(* IEC 61131-3 sources: repolevel_ST_code_completion/output/0127完整版本_带planner/repoeval_Command1/readful_result_no_provide, 10 files *)

(* ---- FB_AirConditioning.st ---- *)
FUNCTION_BLOCK PUBLIC FB_AirConditioning
VAR_OUTPUT
bActive			: BOOL;
lrTemperature	: LREAL;
END_VAR
VAR
lrDefaultTemperature : LREAL := LREAL#0.0; // Explicitly typed initialization
lrCalculatedTemperature : LREAL;
END_VAR

IF bActive THEN
// Calculate the current environment temperature based on control logic
lrCalculatedTemperature := 23.5; // Example fixed value, as logic isn't provided
lrTemperature := lrCalculatedTemperature;
ELSE
// Set temperature to default value when inactive
lrTemperature := lrDefaultTemperature;
END_IF

END_FUNCTION_BLOCK

(* ---- FB_Lamp.st ---- *)
FUNCTION_BLOCK PUBLIC FB_Lamp
VAR_OUTPUT
  byLevel			: BYTE;
END_VAR
VAR
  byNewLevel		: BYTE;
END_VAR

IF byNewLevel > 255 THEN
  byLevel := 255;
ELSE
  byLevel := byNewLevel;
END_IF;
END_FUNCTION_BLOCK

(* ---- FB_Socket.st ---- *)
FUNCTION_BLOCK FB_Socket
VAR_OUTPUT
bActive		: BOOL;
END_VAR
VAR
bInitialized : BOOL := FALSE;
bConnected   : BOOL := FALSE;
END_VAR

IF NOT bInitialized THEN
(* Initialize the socket *)
bInitialized := TRUE;
(* bConnected remains as FALSE; assume not connected initially *)
END_IF

(* Check the connection status *)
IF bInitialized THEN
(* Simulate connection check logic *)
bActive := bConnected;
END_IF

(* Update connection status for the next cycle *)
(* Simulate connection status change logic *)
bConnected := NOT bConnected; (* Toggle connection status for demonstration *)
END_FUNCTION_BLOCK

(* ---- FB_AirConStandbyCommand.st ---- *)
VAR
    bStandbyCommandReceived : BOOL;
    bStandbyConditionsMet : BOOL;
    sExecutionResult : STRING;
END_VAR

bStandbyCommandReceived := FALSE;
bStandbyConditionsMet := FALSE;

// Step 1: Parse input command and check if it is "Standby"
IF __ISVALIDREF(refAirConditioning) THEN
    IF CommandType = "Standby" THEN
        bStandbyCommandReceived := TRUE;
    END_IF;
END_IF;

// Step 2: Check if the air conditioning system can enter standby mode
IF bStandbyCommandReceived THEN
    IF refAirConditioning.bActive AND (refAirConditioning.lrTemperature > 18.0 AND refAirConditioning.lrTemperature < 30.0) THEN
        bStandbyConditionsMet := TRUE;
    END_IF;
END_IF;

// Step 3: Execute standby operation if conditions are met
IF bStandbyConditionsMet THEN
    refAirConditioning.bActive := FALSE;
    sExecutionResult := 'Standby mode activated successfully';
ELSE
    sExecutionResult := 'Failed to activate standby mode';
END_IF;

// Step 4: Update internal system state or necessary flags
IF bStandbyConditionsMet THEN
    SystemState := 'Standby';
ELSE
    SystemState := 'Active';
END_IF;

// Step 5: Output execution result
ExecutionResult := sExecutionResult;
END_FUNCTION_BLOCK

(* ---- FB_CDPlayer.st ---- *)
VAR
	bCurrentState		: BOOL;
	byCurrentVolume		: BYTE;
	byCurrentTrack		: UINT;
END_VAR

IF bPlayerActive THEN
// Update outputs to reflect the current state of the CD player
bPlayerActive := TRUE;
byVolume := byVolume;  // Internal state reflects current volume
byTrack := byTrack;    // Internal state reflects current track
ELSE
// If the player is not active, reset outputs
bPlayerActive := FALSE;
byVolume := 0;
byTrack := 0;
END_IF;
END_FUNCTION_BLOCK

(* ---- FB_LampSetLevelCommand.st ---- *)
VAR
	refLamp		: REFERENCE TO FB_Lamp;
	byNewLevel	: BYTE;
	bResult		: BOOL;
END_VAR

IF (__ISVALIDREF(refLamp)) THEN
 IF (byNewLevel > 100) THEN
  byNewLevel := 100; // Set to maximum allowed value if out of range
 END_IF

 // BYTE data type cannot be less than 0, so no check for values < 0 is needed.

 bResult := refLamp.SetLevel(byNewLevel); // Update brightness level in hardware

 IF bResult THEN
  RETURN; // Command executed successfully
 END_IF
END_IF

bResult := FALSE; // Command execution failed
RETURN;
END_FUNCTION_BLOCK

(* ---- FB_MusicPlayCommand.st ---- *)
VAR
    isCommandActive : BOOL; // Indicates if the play command is active
    isPlaying : BOOL; // Indicates if music is currently playing
    errorStatus : BOOL; // Indicates if there was an error during execution
    logTimestamp : TIME; // Stores the timestamp of the last successful execution
END_VAR

IF NOT isCommandActive THEN
    RETURN;
END_IF;

IF __ISVALIDREF(refCDPlayer) THEN
    refCDPlayer.Start();
    IF refCDPlayer.IsPlaying THEN
        isPlaying := TRUE;
        errorStatus := FALSE;
logTimestamp := T#0s; // Assign placeholder timestamp value since CURRENT_TIME is invalid
    ELSE
        isPlaying := FALSE;
        errorStatus := TRUE;
    END_IF;
ELSE
    errorStatus := TRUE;
END_IF;
END_FUNCTION_BLOCK

(* ---- FB_SocketOffCommand.st ---- *)
VAR
    bCommandExecuted : BOOL := FALSE;
END_VAR

IF NOT bCommandExecuted THEN
    (* Step 1: Initialize command state *)
    bCommandExecuted := TRUE;

    (* Step 2: Call control logic to turn off the socket *)
    IF __ISVALIDREF(THIS^.refSocket) THEN
        THIS^.refSocket.Off();
    END_IF;

    (* Step 3: Update socket state to off *)
    IF __ISVALIDREF(THIS^.refSocket) THEN
        THIS^.refSocket.bActive := FALSE;
    END_IF;

    (* Step 4: Indicate command execution success *)
    bCommandExecuted := TRUE;
END_IF;

(* Step 5: Clean up resources if necessary *)
(* No additional resources to clean up in this implementation *)
END_FUNCTION_BLOCK

(* ---- FB_SocketOnCommand.st ---- *)
VAR
    refSocket : REFERENCE TO FB_Socket;
    bCommandValid : BOOL;
END_VAR

VAR_INPUT
    sCommand : STRING;
END_VAR

VAR_OUTPUT
    bSuccess : BOOL;
    sErrorMessage : STRING;
END_VAR

VAR
    bSocketState : BOOL;
END_VAR

// Implementation
IF NOT __ISVALIDREF(refSocket) THEN
 bSuccess := FALSE; // Mark the operation as unsuccessful.
 sErrorMessage := 'Invalid socket reference'; // Provide an error message for debugging.
 RETURN; // Exit the function block to avoid further invalid operations.
END_IF

// Step 1: Initialize internal state variables
bCommandValid := FALSE; // State validity flag for the command, starts invalid.

// Step 2: Parse the command
IF sCommand = 'ON' THEN
  bCommandValid := TRUE; // Command recognized as valid for turning ON.
  bSocketState := TRUE;  // Set socket state to ON.
ELSIF sCommand = 'OFF' THEN
  bCommandValid := TRUE; // Command recognized as valid for turning OFF.
  bSocketState := FALSE; // Set socket state to OFF.
ELSE
  bCommandValid := FALSE; // Invalid command received; set validation to FALSE.
END_IF

// Step 3: Validate command parameters
IF NOT bCommandValid THEN
    bSuccess := FALSE;
    sErrorMessage := 'Invalid command';
    RETURN;
END_IF

// Step 4: Control the socket
IF bSocketState THEN
refSocket.On(); // Turns the socket ON correctly. Verify that the 'On' method is implemented in the FB_Socket block.
ELSE
refSocket.Off(); // Turns the socket OFF correctly. Verify that the 'Off' method is implemented in the FB_Socket block.
END_IF

// Step 5: Set output status
bSuccess := TRUE; // Operation completed successfully.
sErrorMessage := ''; // Clear any prior error messages.

// Step 6: Handle exceptions (already handled in validation steps above)
RETURN;
END_FUNCTION_BLOCK

(* ---- FB_SwitchPanel.st ---- *)
VAR
	aiCommand		: ARRAY[1..8] OF I_Command;
	arrRtrig		: ARRAY[1..8] OF R_TRIG;
	nIndex			: INT;
END_VAR

FOR nIndex := 1 TO 8 DO
	arrRtrig[nIndex](CLK := arrSwitch[nIndex]);
	IF arrRtrig[nIndex].Q THEN
IF aiCommand[nIndex].Valid THEN // Assuming 'Valid' is a method or property to check usability
   aiCommand[nIndex](Execute := TRUE);
END_IF
	END_IF
END_FOR
END_FUNCTION_BLOCK
